# EPICS IOC start-up script: iocsh/ethercatmcAnalogInput-TSE.iocsh
ethercatmcCreateAsynParam $(MOTOR_PORT) $(ASYNPARAMNAME)      Float64

dbLoadRecords("ethercatmcAnalogInput.template", "P=$(P), R=$(R), MOTOR_PORT=$(MOTOR_PORT), CHNO=$(CHNO), ASYNPARAMNAME=$(ASYNPARAMNAME), PREC=$(PREC), DESC=$(DESC), EGU=$(EGU), TSE=$(TSE)")
